// LS Electric XG5000 project: DELXGHS
// PLC LSPLC

PROGRAM NewProgram (task: 스캔 프로그램)

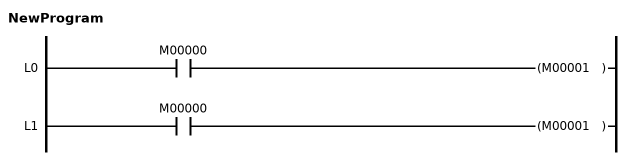
; L0
// network not rendered as a mnemonic list; see the picture
; L1
LOAD      M00000
OUT       M00001